(* CODESYS project SP5IOtest.project

Project tree, tasks and I/O mapping:
  Device : Owen SPK2xx 03.CS.WEB, Owen, order no. 023, version 3.5.4.20
    application Application
      libraries: Standard, * (System); VisuDialogs, * (System); CmpSysExec, 1.0.0.2 (Owen); SPK_Tools, 1.0.1 (Owen); RS mode library, 1.0.0.0 (Owen); ArchiverSPK, 3.5.3.53 (Owen); CAA File, 3.5.5.0 (CAA Technical Workgroup)
      task MainTask (cyclic, interval t#10ms, priority 1) calls PLC_PRG
      task VISU_TASK (cyclic, interval 10 ms, priority 30) calls VisuElems.Visu_Prg
      program PLC_PRG [ST]
      visualisation Visualization
      global variables GVL
      visualisation ManualInput
      image pool ImagePool
      visualisation Settings
      data type TableStruct
      visualisation ArrayTest
      RecipeManager
        recipe definition Receipt: PLC_PRG.arrayOfIngr[0].nameOfIngr : STRING; PLC_PRG.arrayOfIngr[0].weightOfIngr : STRING; PLC_PRG.arrayOfIngr[0].isDissolve : STRING; PLC_PRG.arrayOfIngr[0].timeOfMixing : STRING; PLC_PRG.arrayOfIngr[0].addMessage : STRING; PLC_PRG.arrayOfIngr[1].nameOfIngr : STRING; PLC_PRG.arrayOfIngr[1].weightOfIngr : STRING; PLC_PRG.arrayOfIngr[1].isDissolve : STRING; PLC_PRG.arrayOfIngr[1].timeOfMixing : STRING; PLC_PRG.arrayOfIngr[1].addMessage : STRING; PLC_PRG.arrayOfIngr[2].nameOfIngr : STRING; PLC_PRG.arrayOfIngr[2].weightOfIngr : STRING; PLC_PRG.arrayOfIngr[2].isDissolve : STRING; PLC_PRG.arrayOfIngr[2].timeOfMixing : STRING; PLC_PRG.arrayOfIngr[2].addMessage : STRING; PLC_PRG.arrayOfIngr[3].nameOfIngr : STRING; PLC_PRG.arrayOfIngr[3].weightOfIngr : STRING; PLC_PRG.arrayOfIngr[3].isDissolve : STRING; PLC_PRG.arrayOfIngr[3].timeOfMixing : STRING; PLC_PRG.arrayOfIngr[3].addMessage : STRING; PLC_PRG.arrayOfIngr[4].nameOfIngr : STRING; PLC_PRG.arrayOfIngr[4].weightOfIngr : STRING; PLC_PRG.arrayOfIngr[4].isDissolve : STRING; PLC_PRG.arrayOfIngr[4].timeOfMixing : STRING; PLC_PRG.arrayOfIngr[4].addMessage : STRING; PLC_PRG.arrayOfIngr[5].nameOfIngr : STRING; PLC_PRG.arrayOfIngr[5].weightOfIngr : STRING; PLC_PRG.arrayOfIngr[5].isDissolve : STRING; PLC_PRG.arrayOfIngr[5].timeOfMixing : STRING; PLC_PRG.arrayOfIngr[5].addMessage : STRING; PLC_PRG.arrayOfIngr[6].nameOfIngr : STRING; PLC_PRG.arrayOfIngr[6].weightOfIngr : STRING; PLC_PRG.arrayOfIngr[6].isDissolve : STRING; PLC_PRG.arrayOfIngr[6].timeOfMixing : STRING; PLC_PRG.arrayOfIngr[6].addMessage : STRING; PLC_PRG.arrayOfIngr[7].nameOfIngr : STRING; PLC_PRG.arrayOfIngr[7].weightOfIngr : STRING; PLC_PRG.arrayOfIngr[7].isDissolve : STRING; PLC_PRG.arrayOfIngr[7].timeOfMixing : STRING; PLC_PRG.arrayOfIngr[7].addMessage : STRING; PLC_PRG.arrayOfIngr[8].nameOfIngr : STRING; PLC_PRG.arrayOfIngr[8].weightOfIngr : STRING; PLC_PRG.arrayOfIngr[8].isDissolve : STRING; PLC_PRG.arrayOfIngr[8].timeOfMixing : STRING; PLC_PRG.arrayOfIngr[8].addMessage : STRING; PLC_PRG.arrayOfIngr[9].nameOfIngr : STRING; PLC_PRG.arrayOfIngr[9].weightOfIngr : STRING; PLC_PRG.arrayOfIngr[9].isDissolve : STRING; PLC_PRG.arrayOfIngr[9].timeOfMixing : STRING; PLC_PRG.arrayOfIngr[9].addMessage : STRING; PLC_PRG.arrayOfIngr[10].nameOfIngr : STRING; PLC_PRG.arrayOfIngr[10].weightOfIngr : STRING; PLC_PRG.arrayOfIngr[10].isDissolve : STRING; PLC_PRG.arrayOfIngr[10].timeOfMixing : STRING; PLC_PRG.arrayOfIngr[10].addMessage : STRING
      function two_word_to_real [ST]
      function block FileReciple [ST]
    Modbus_COM : Modbus COM, 3S - Smart Software Solutions GmbH, version 3.4.0.0
        settings: DataBits = 8; StopBits = 1; ComPort = 3
      Modbus_Master_COM_Port : Modbus Master, COM Port, 3S - Smart Software Solutions GmbH, version 3.5.5.0
          settings: Transmission = 'RTU'; ResponseTimeout = 300; TimeBetweenFrames = 50; Auto-restart communication = TRUE
        Modbus_Slave_COM_Port : Modbus Slave, COM Port, 3S - Smart Software Solutions GmbH, version 3.5.4.0
            settings: SlaveAddress = 16; ResponseTimeout = 300; UseExtendedFunctionCodes = TRUE; Channel 1.Function Code = 16; Channel 1.Read Offset = 0; Channel 1.Read Length = 0; Channel 1.Write Offset = 16#0032; Channel 1.Write Length = 1; Channel 1.Cycle Time = 100
            output Application.outputDiscrets : WORD  // Channel 1.Channel 1[0]
            unmapped channels: Channel 1
    Modbus_COM_1 : Modbus COM, 3S - Smart Software Solutions GmbH, version 3.4.0.0
        settings: DataBits = 8; StopBits = 1; ComPort = 4
      Modbus_Master_COM_Port_1 : Modbus Master, COM Port, 3S - Smart Software Solutions GmbH, version 3.5.5.0
          settings: Transmission = 'RTU'; ResponseTimeout = 300; TimeBetweenFrames = 50; Auto-restart communication = TRUE
        Modbus_Slave_COM_Port_1 : Modbus Slave, COM Port, 3S - Smart Software Solutions GmbH, version 3.5.4.0
            settings: SlaveAddress = 32; ResponseTimeout = 300; UseExtendedFunctionCodes = TRUE; Channel 1.Function Code = 3; Channel 1.Read Offset = 16#0046; Channel 1.Read Length = 2; Channel 1.Write Offset = 0; Channel 1.Write Length = 0; Channel 1.Cycle Time = 100; Channel 2.Function Code = 3; Channel 2.Read Offset = 16#0048; Channel 2.Read Length = 2; Channel 2.Write Offset = 0; Channel 2.Write Length = 0; Channel 2.Cycle Time = 100; Channel 3.Function Code = 3; Channel 3.Read Offset = 16#004A; Channel 3.Read Length = 2; Channel 3.Write Offset = 0; Channel 3.Write Length = 0; Channel 3.Cycle Time = 100; Channel 4.Function Code = 3; Channel 4.Read Offset = 16#004C; Channel 4.Read Length = 2; Channel 4.Write Offset = 0; Channel 4.Write Length = 0; Channel 4.Cycle Time = 100
            input  Application.arr1[0] : WORD  // Channel 1.Channel 1
            input  Application.arr1[1] : WORD  // Channel 1.Channel 1
            input  Application.arr2[0] : WORD  // Channel 2.Channel 2
            input  Application.arr2[1] : WORD  // Channel 2.Channel 2
            input  Application.arr3[0] : WORD  // Channel 3.Channel 3
            input  Application.arr3[1] : WORD  // Channel 3.Channel 3
            input  Application.arr4[0] : WORD  // Channel 4.Channel 4
            input  Application.arr4[1] : WORD  // Channel 4.Channel 4
            unmapped channels: Channel 1, Channel 2, Channel 3, Channel 4
  text list GlobalTextList
  GlobalImagePool
  image pool ImagePool
  5ce3da45-db07-42e7-a21c-a00fff4ed8f6|C:\Users\Валентин\Desktop\home.png
  5ce3da45-db07-42e7-a21c-a00fff4ed8f6|D:\Pictures\tanzania.jpg
  5ce3da45-db07-42e7-a21c-a00fff4ed8f6|D:\Pictures\tanzania800x480.jpg
  5ce3da45-db07-42e7-a21c-a00fff4ed8f6|D:\Pictures\BeachHouse800x480.jpg
  5ce3da45-db07-42e7-a21c-a00fff4ed8f6|D:\Projects\OWEN\JAVA\GIT\settings.png
  5ce3da45-db07-42e7-a21c-a00fff4ed8f6|D:\Projects\OWEN\PIC\motherboard.png
  5ce3da45-db07-42e7-a21c-a00fff4ed8f6|D:\Projects\OWEN\PIC\home.png
  5ce3da45-db07-42e7-a21c-a00fff4ed8f6|D:\Projects\OWEN\PIC\settings.jpg
  5ce3da45-db07-42e7-a21c-a00fff4ed8f6|D:\Projects\OWEN\PIC\reset.jpg
  5ce3da45-db07-42e7-a21c-a00fff4ed8f6|D:\Projects\OWEN\PIC\reset.png
  5ce3da45-db07-42e7-a21c-a00fff4ed8f6|D:\Projects\OWEN\PIC\resetButton.png
  5ce3da45-db07-42e7-a21c-a00fff4ed8f6|D:\Projects\OWEN\PIC\start.png
  5ce3da45-db07-42e7-a21c-a00fff4ed8f6|D:\Projects\OWEN\PIC\remove.png
  5ce3da45-db07-42e7-a21c-a00fff4ed8f6|D:\Projects\OWEN\PIC\ok.png
  5ce3da45-db07-42e7-a21c-a00fff4ed8f6|D:\Projects\OWEN\PIC\cancel.png
  function block Time_Struct [ST]
  5ce3da45-db07-42e7-a21c-a00fff4ed8f6|D:\Projects\OWEN\PIC\add.png
  5ce3da45-db07-42e7-a21c-a00fff4ed8f6|D:\Projects\OWEN\PIC\back.png
  5ce3da45-db07-42e7-a21c-a00fff4ed8f6|D:\Projects\OWEN\PIC\next.png
  5ce3da45-db07-42e7-a21c-a00fff4ed8f6|D:\Projects\OWEN\PIC\Drives-Downloads-icon.png
  5ce3da45-db07-42e7-a21c-a00fff4ed8f6|D:\Projects\OWEN\PIC\Actions-application-exit-icon.png
  5ce3da45-db07-42e7-a21c-a00fff4ed8f6|D:\Projects\OWEN\PIC\App-desktop-enhancements-icon.png
  5ce3da45-db07-42e7-a21c-a00fff4ed8f6|D:\Projects\OWEN\PIC\chemistryS.png
  5ce3da45-db07-42e7-a21c-a00fff4ed8f6|D:\Projects\OWEN\PIC\chemistry.png
  5ce3da45-db07-42e7-a21c-a00fff4ed8f6|D:\Projects\OWEN\PIC\Iconshock-Real-Vista-Education-Laboratory.png
*)

// Device/Application/TableStruct
TYPE TableStruct :
STRUCT
	nameOfIngr:STRING;
	weightOfIngr:STRING;
	isDissolve:STRING;
	timeOfMixing:STRING;
	addMessage:STRING;
	
END_STRUCT
END_TYPE

// Device/Application/GVL
VAR_GLOBAL
	outputDiscrets: INT;
	arr1:ARRAY[0..1]OF WORD;		
	arr2:ARRAY[0..1]OF WORD;
	arr3:ARRAY[0..1]OF WORD;
	arr4:ARRAY[0..1]OF WORD;
	
END_VAR

// Device/Application/PLC_PRG
PROGRAM PLC_PRG
VAR
	down: STRING;
	
	
	resipeExt: STRING :='Receipt';
	RecipeManCommands 		: RecipeManCommands;
//----------------------------------------------------------------\\	
	data0:real;
	data1:WORD;
	download:BOOL;
	save:BOOL;
	ingrArrayLength: INT := 10;
	arrayOfIngr: ARRAY[0..10] OF TableStruct;
	FileRec:FileReciple(FileName:='Recipe.txt', pr:=ADR(arrayOfIngr),size:=SIZEOF(arrayOfIngr));
	x: INT := 0;
	edge: INT := 1000;
	light: BOOL;
	swich: BOOL;	
	lamp1: BOOL := outputDiscrets.0;
	increment: INT := 1;	
	manualButtonStart: BOOL;
	testButton: BOOL;
	cleanCounter:INT;
	strings: ARRAY[0..1] OF STRING := ['zero', 'one'];
	fileLoader: BOOL;
END_VAR
VAR RETAIN
	list: STRING:='List';
	file: STRING:='';
	writeToTable:BOOL;
	idxOfLine:INT := 0;
	currentPrgName: STRING;
	fileName: STRING;
	currentIngredientName: STRING;
	currentTimeMixing: TIME;
	maximumWeight: INT := 1000;
	currentWeight: INT;
	currentPoint : INT;
	manualMode: BOOL;
	dissolve: BOOL;
	message: STRING;
END_VAR

data0:=two_word_to_real(ADR(arr1));
data1:=arr1[1];
IF lamp1 = TRUE THEN
	outputDiscrets.0:=TRUE;
	ELSE
	outputDiscrets.0:=FALSE;
END_IF
IF writeTotable = TRUE THEN
	arrayOfIngr[idxOfLine].nameOfIngr:=currentIngredientName;
	arrayOfIngr[idxOfLine].weightOfIngr:=INT_TO_STRING(currentWeight);
	arrayOfIngr[idxOfLine].isDissolve:=BOOL_TO_STRING(dissolve);
	arrayOfIngr[idxOfLine].timeOfMixing:=TIME_TO_STRING(currentTimeMixing);
	arrayOfIngr[idxOfLine].addMessage:=message;
	idxOfLine := idxOfLine + 1;		
	writeTotable:=FALSE;
	IF idxOfLine > ingrArrayLength THEN
		idxOfLine := 0;
	END_IF
END_IF

IF fileLoader = TRUE THEN
	fileName:=concat(currentPrgName,'.Receipt.txt');	
	RecipeManCommands.LoadFromAndWriteRecipe('Receipt', currentPrgName, fileName);
	fileLoader := FALSE;
	down:= 'Pressed';
END_IF

IF swich = TRUE THEN
x := x + increment;
light := TRUE;
 IF x >= currentWeight + currentPoint THEN 
	 currentPoint:= currentPoint+currentWeight;
	 increment:=0;
 outputDiscrets.0:=TRUE; 
 swich:= FALSE; 
 END_IF	 		
END_IF

IF manualMode = TRUE THEN
	swich:=TRUE;
END_IF

END_PROGRAM

// Device/Application/two_word_to_real
FUNCTION two_word_to_real : REAL
VAR_INPUT
	in_data: POINTER TO ARRAY[0..1]OF WORD;
END_VAR
VAR
	p1:POINTER TO BYTE;
	p2:pointer to byte;
END_VAR

p1:=ADR(two_word_to_real);
p2:=ADR(in_data^[1]);

p1^:=p2^;
p1:=p1+1;
p2:=p2+1;
p1^:=p2^;
p1:=p1+1;
p2:=ADR(in_data^[0]);
p1^:=p2^;
p1:=p1+1;
p2:=p2+1;
p1^:=p2^;

END_FUNCTION

// Device/Application/FileReciple
FUNCTION_BLOCK FileReciple
VAR_INPUT
	FileName: STRING(15);    (*Имя файла с рецептами*)
    pt:    POINTER    TO ARRAY [0..32000] OF TableStruct;    (*Указатель на массив с рецептами*)
    size:UINT;    (*Размер массива рецептов*)
    Restore: BOOL;    (*Загрузить рецепты из файла*)
    Save: BOOL;    (*Сохранить рецепты в файл*)
END_VAR
VAR_OUTPUT
END_VAR
VAR
	
	StatusOfFile: INT:=100;    (*Это значение нужно для правильной инициализации ФБ*)
    f: DWORD;    (*Дескриптор файла*)
    statusf: DWORD;
    NULL:TableStruct;    (*Пустая запись в массиве рецептов*)
    i: INT;
    R_TRIG1: R_TRIG;
    R_TRIG2: R_TRIG;
    f_err: BOOL;
END_VAR

CASE StatusOfFile OF
0:
    R_TRIG1(CLK:=Restore);
    R_TRIG2(CLK:=Save);
    IF    R_TRIG1.Q    THEN
        StatusOfFile:=100;    (*Восстановить рецепты из файла*)
    END_IF
    IF    R_TRIG2.Q    THEN
        StatusOfFile:=8;    (*Записать рецепты в файл*)
    END_IF

8:    (*Удалить старую версию файла .bak*)
    f_err:=File.Delete(CONCAT(FileName, '.bak'));StatusOfFile:=10;


10:    (*сохранить новую версию файла .bak*)
    statusf:=File.Copy(CONCAT(FileName, '.bak'), FileName);StatusOfFile:=11;


11:    (*открыть файл на запись*)
    f:=File.Open(FileName, 'w');StatusOfFile:=12;


12:    (*записать рецепты в файл*)
    statusf:=File.Write(f, pt, size);StatusOfFile:=102;


(*Эта часть выполняется однократно после старта ПЛК*)
100: (*Открыть файл на чтение*)
    f:=File.Open(FileName, 'r');
    IF f=0 THEN
        StatusOfFile:=200; (*Нет такого файла*)
    ELSE
        StatusOfFile:=101;    (*ОК, файл существует*)
    END_IF


101: (*Прочитать файл в массив рецептов*)
    statusf:=File.Read(f, pt, size);StatusOfFile:=102;


102: (*Закрываем файл*)
    File.Close(f);StatusOfFile:=103;


103:    (*Конец инициализации после включения ПЛК*)
        StatusOfFile:=0;


200: (*Если файла нет, то попробовать его восстановить*)
    statusf:=File.Copy(FileName, CONCAT(FileName, '.bak'));StatusOfFile:=201;


201:
    IF statusf=0 THEN (*старой версии файла нет, создать новый пустой файл*)
        FOR i:=0    TO size/SIZEOF(NULL)-1    DO
            NULL.nameOfIngr:=CONCAT('Набор_', INT_TO_STRING(i+1));
            pt^[i]:=NULL;
        END_FOR
        StatusOfFile:=11; (*Записать новый файл*)
    ELSE
        StatusOfFile:=100;
    END_IF
END_CASE

END_FUNCTION_BLOCK

// Time_Struct
FUNCTION_BLOCK Time_Struct
VAR_INPUT
	Type_Time:TIME;
END_VAR
VAR_OUTPUT
	Day:DWORD;
	Hour:DWORD;
	Minute:DWORD;
	Second:DWORD;
	Millisecond:DWORD;  
END_VAR
VAR
		Time_DWORD:DWORD;
		Day_Ost:DWORD;
		Hour_Ost:DWORD;
		Minute_Ost:DWORD;
		Second_Ost:DWORD;
		Millisecond_Ost:DWORD; 
END_VAR


Time_DWORD := TIME_TO_DWORD(Type_Time);

Millisecond := Second_Ost;

Second := Minute_Ost/ 1000;
Second_Ost := Minute_Ost MOD 1000;

Minute := Hour_Ost/60000;
Minute_Ost := Hour_Ost MOD 60000;

Hour := Day_Ost/3600000;
Hour_Ost := Day_Ost MOD 3600000;

Day := Time_DWORD/86400000;
Day_Ost := Time_DWORD MOD 86400000;

END_FUNCTION_BLOCK

// Device/Application/Visualization
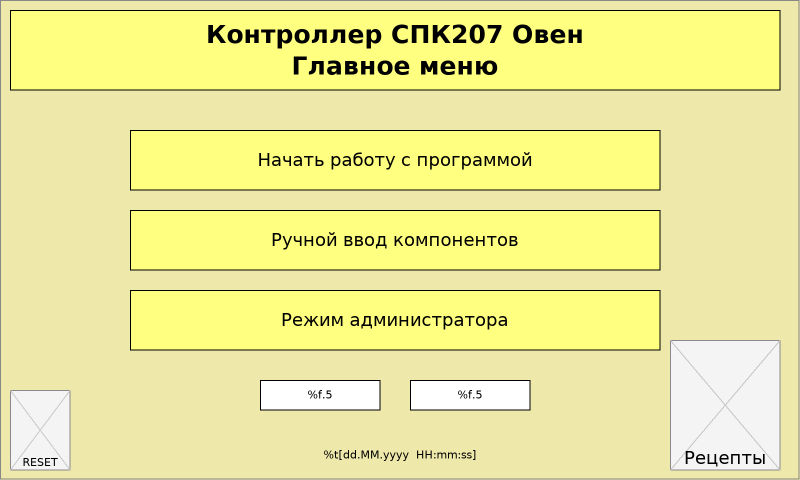
VISUALIZATION Visualization  // 800x480
    Image (10,390 60x80), "RESET", image: ImagePool.start
        OnMouseClick: execute {
            //SysExecute('/sbin/reboot');
        }
    Image (670,340 110x130), "Рецепты", image: ImagePool.Iconshock-Real-Vista-Education-Laboratory
        OnMouseClick:  Assign=Settings, Type=Assignment
    RoundedRectangle (10,10 770x80), "Контроллер СПК207 Овен Главное меню"
    RoundedRectangle (130,130 530x60), "Начать работу с программой"
    RoundedRectangle (130,210 530x60), "Ручной ввод компонентов"
        OnMouseClick:  Assign=ManualInput, Type=Assignment
        OnMouseClick: execute { PLC_PRG.manualMode:=true; }
    RoundedRectangle (130,290 530x60), "Режим администратора"
        OnMouseClick:  Type=Login
    Rectangle (300,440 200x30), "%t[dd.MM.yyyy HH:mm:ss]"
    RoundedRectangle (260,380 120x30), "%f.5", text variable: PLC_PRG.data0
    RoundedRectangle (410,380 120x30), "%f.5", text variable: PLC_PRG.data1
END_VISUALIZATION

// Device/Application/ManualInput
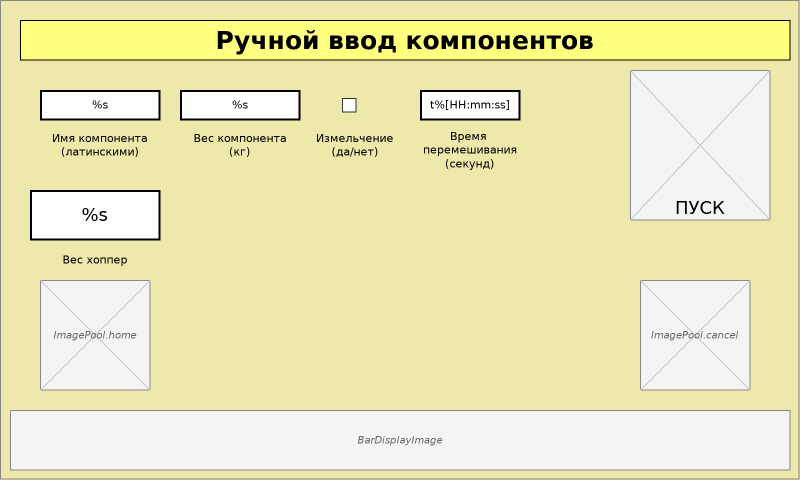
VISUALIZATION ManualInput  // 800x480
    RoundedRectangle (20,20 770x40), "Ручной ввод компонентов"
    RoundedRectangle (180,90 120x30), "%s", text variable: PLC_PRG.currentWeight
        OnMouseClick: execute { PLC_PRG.edge:=PLC_PRG.maximumWeight -PLC_PRG.x; }
        OnMouseClick: write PLC_PRG.currentWeight via VisuDialogs.Numpad, min 10, max PLC_PRG.edge
    RoundedRectangle (180,130 120x30), "Вес компонента (кг)"
    RoundedRectangle (300,130 110x30), "Измельчение (да/нет)"
    RoundedRectangle (420,90 100x30), "t%[HH:mm:ss]", colour toggle: PLC_PRG.testButton
        OnMouseClick: write the text variable via VisuDialogs.Numpad
    RoundedRectangle (400,130 140x40), "Время перемешивания (секунд)"
    Image (630,70 140x150), "ПУСК", image: ImagePool.ok
        OnMouseClick:  ToggleVariable=PLC_PRG.swich
        OnMouseClick: execute {
            IF PLC_PRG.currentWeight > 0
            THEN PLC_PRG.increment:=1;
            END_IF
        }
    BarDisplayImage (10,410 780x60), value: PLC_PRG.x, style: BarDisplayImage-Gray, scale format: %.0f, scale 0..1000
    RoundedRectangle (30,190 130x50), "%s", text variable: PLC_PRG.x
        OnMouseClick: execute { PLC_PRG.edge:=PLC_PRG.maximumWeight -PLC_PRG.x; }
        OnMouseClick: write PLC_PRG.currentWeight via VisuDialogs.Numpad, min 10, max PLC_PRG.edge
    Image (40,280 110x110), image: ImagePool.home
        OnMouseClick:  Assign=Visualization, Type=Assignment
        OnMouseClick: execute { PLC_PRG.manualMode:=false; }
    Image (640,280 110x110), image: ImagePool.cancel
        OnMouseClick: execute {
            PLC_PRG.x:=0;
            PLC_PRG.currentWeight:=0;
            PLC_PRG.currentPoint:=0;
        }
    RoundedRectangle (40,90 120x30), "%s", text variable: PLC_PRG.currentIngredientName
        OnMouseClick: write the text variable via VisuDialogs.Keypad, min 1, max 30
    RoundedRectangle (40,130 120x30), "Имя компонента (латинскими)"
    RoundedRectangle (30,250 130x20), "Вес хоппер"
    Checkbox (340,90 30x30), variable: PLC_PRG.dissolve
END_VISUALIZATION

// Device/Application/Settings
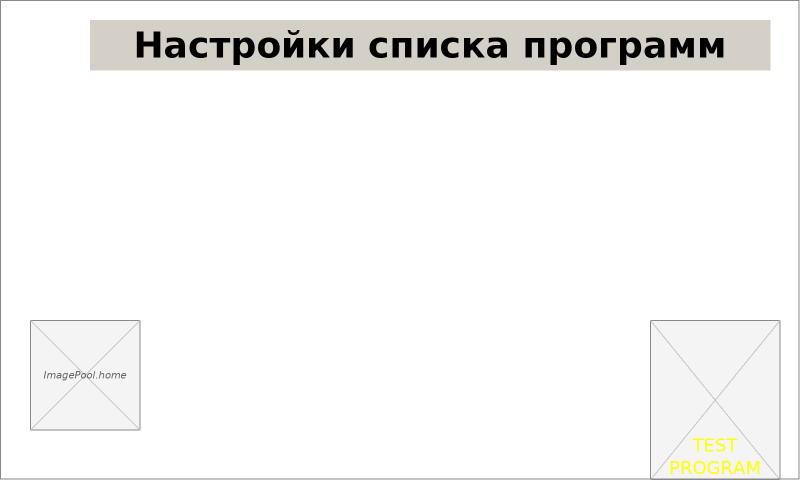
VISUALIZATION Settings  // 800x480, background image ImagePool.settings0
    Rectangle (90,20 680x50), "Настройки списка программ"
    Image (30,320 110x110), image: ImagePool.home
        OnMouseClick:  Assign=Visualization, Type=Assignment
    Image (650,320 130x160), "TEST PROGRAM", image: ImagePool.next
        OnMouseClick:  Assign=ArrayTest, Type=Assignment
END_VISUALIZATION

// Device/Application/ArrayTest
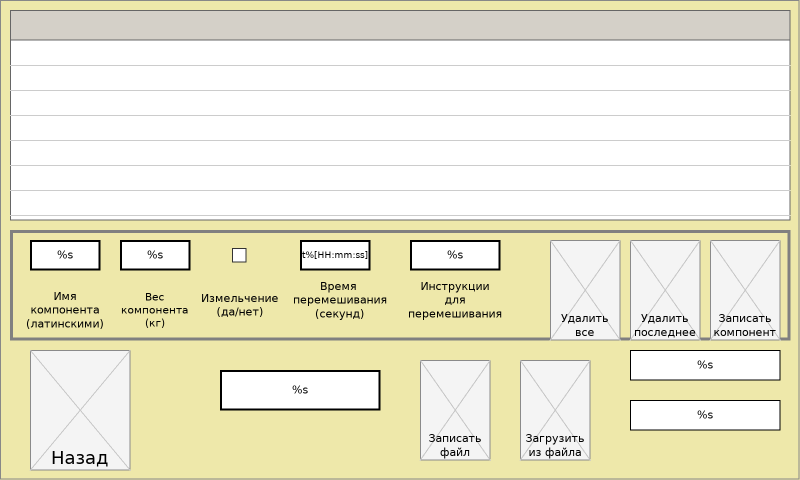
VISUALIZATION ArrayTest  // 800x480
    Rectangle (10,230 780x110)
    Table (10,10 780x210), data array: PLC_PRG.arrayOfIngr
        p1128707560: PLC_PRG.ingrArrayLength
        p3854506369: PLC_PRG.arrayOfIngr[INDEX].nameOfIngr
        p1892666644: PLC_PRG.arrayOfIngr[INDEX].weightOfIngr
        p338671338: PLC_PRG.arrayOfIngr[INDEX].isDissolve
        p2170511999: PLC_PRG.arrayOfIngr[INDEX].timeOfMixing
        p3723444502: PLC_PRG.arrayOfIngr[INDEX].addMessage
        p2232123230: Name of the ingredient
        p1755163831: is dissolve
    RoundedRectangle (120,240 70x30), "%s", text variable: PLC_PRG.currentWeight
        OnMouseClick: execute { PLC_PRG.edge:=PLC_PRG.maximumWeight -PLC_PRG.x; }
        OnMouseClick: write PLC_PRG.currentWeight via VisuDialogs.Numpad, min 10, max PLC_PRG.edge
    RoundedRectangle (120,280 70x60), "Вес компонента (кг)"
    RoundedRectangle (200,280 80x50), "Измельчение (да/нет)"
    RoundedRectangle (300,240 70x30), "t%[HH:mm:ss]", text variable: PLC_PRG.currentTimeMixing, colour toggle: PLC_PRG.testButton
        OnMouseClick: write the text variable via VisuDialogs.Numpad
    RoundedRectangle (290,280 100x40), "Время перемешивания (секунд)"
    RoundedRectangle (30,240 70x30), "%s", text variable: PLC_PRG.currentIngredientName
        OnMouseClick: write the text variable via VisuDialogs.Keypad, min 1, max 30
    RoundedRectangle (20,280 90x60), "Имя компонента (латинскими)"
    Checkbox (230,240 30x30), variable: PLC_PRG.dissolve
    Image (550,240 70x100), "Удалить все", image: ImagePool.cancel
        OnMouseClick: execute {
            FOR PLC_PRG.cleanCounter:=0 TO PLC_PRG.ingrArrayLength DO
            	PLC_PRG.arrayOfIngr[PLC_PRG.cleanCounter].nameOfIngr:='';
            	PLC_PRG.arrayOfIngr[PLC_PRG.cleanCounter].weightOfIngr:='';
            	PLC_PRG.arrayOfIngr[PLC_PRG.cleanCounter].isDissolve:='';
            	PLC_PRG.arrayOfIngr[PLC_PRG.cleanCounter].timeOfMixing:='';
            	PLC_PRG.arrayOfIngr[PLC_PRG.cleanCounter].addMessage:='';
            END_FOR
             PLC_PRG.cleanCounter:=0;
             PLC_PRG.idxOfLine:=0;
        }
    Image (630,240 70x100), "Удалить последнее", image: ImagePool.remove
        OnMouseClick: execute {
            IF PLC_PRG.idxOfLine > 0 THEN
             PLC_PRG.idxOfLine:=PLC_PRG.idxOfLine - 1;
             END_IF
            	PLC_PRG.arrayOfIngr[PLC_PRG.idxOfLine].nameOfIngr:='';
            	PLC_PRG.arrayOfIngr[PLC_PRG.idxOfLine].weightOfIngr:='';
            	PLC_PRG.arrayOfIngr[PLC_PRG.idxOfLine].isDissolve:='';
            	PLC_PRG.arrayOfIngr[PLC_PRG.idxOfLine].timeOfMixing:='';
            	PLC_PRG.arrayOfIngr[PLC_PRG.idxOfLine].addMessage:='';
        }
    Image (710,240 70x100), "Записать компонент", image: ImagePool.add
        OnMouseClick:  ToggleVariable=PLC_PRG.writeToTable
    Image (30,350 100x120), "Назад", image: ImagePool.back
        OnMouseClick:  Assign=Settings, Type=Assignment
    RoundedRectangle (410,240 90x30), "%s", text variable: PLC_PRG.message
        OnMouseClick: write the text variable via VisuDialogs.Keypad, min 1, max 30
    RoundedRectangle (400,280 110x40), "Инструкции для перемешивания"
    Image (420,360 70x100), "Записать файл", image: ImagePool.Drives-Downloads-icon
        OnMouseClick: execute { PLC_PRG.RecipeManCommands.CreateRecipe(PLC_PRG.resipeExt,PLC_PRG.currentPrgName); }
    Image (520,360 70x100), "Загрузить из файла", image: ImagePool.App-desktop-enhancements-icon
        OnMouseClick:  ToggleVariable=PLC_PRG.fileLoader
    RoundedRectangle (220,370 160x40), "%s", text variable: PLC_PRG.currentPrgName
        OnMouseClick: write the text variable via VisuDialogs.Keypad, min 1, max 30
    Rectangle (630,350 150x30), "%s", text variable: PLC_PRG.down
    Rectangle (630,400 150x30), "%s", text variable: PLC_PRG.fileName
END_VISUALIZATION
